// TwinCAT 3 PLC project Sample02
// ProgramVersion: 3.1.4020.10
// libraries:
//   Tc2_Standard, * (Beckhoff Automation GmbH)
//   Tc2_System, * (Beckhoff Automation GmbH)
//   Tc3_Module, * (Beckhoff Automation GmbH)
// project tree:
//   / PlcTask.TcTTO (not stored)
//   POUs/ Class Diagram.TcCD (not stored), FB_AnalogValue.TcPOU, FB_Controller.TcPOU, FB_Lamp.TcPOU, FB_LampUpDown.TcPOU, FB_LampSetDirect.TcPOU, FB_LampOnOff.TcPOU, I_Lamp.TcIO, I_Observer.TcIO, I_Subject.TcIO, MAIN.TcPOU
// real-time tasks:
//   TASK PlcTask: cycle T#10ms, priority 20, ADS port 350

// ---- POUs/I_Lamp.TcIO
INTERFACE I_Lamp

// Reduces the control value by 5 in the range of 10 to 100.
METHOD DimDown
VAR_INPUT
END_VAR
END_METHOD

// Increments the control value by 5 in the range of 10 to 100.
METHOD DimUp
VAR_INPUT
END_VAR
END_METHOD

// Sets the control value to 0.
METHOD Off
VAR_INPUT
END_VAR
END_METHOD

// Sets the control value to 100.
METHOD On
VAR_INPUT
END_VAR
END_METHOD

END_INTERFACE

// ---- POUs/I_Observer.TcIO
INTERFACE I_Observer EXTENDS __System.IQueryInterface

METHOD Update : BYTE
VAR_INPUT
	nNewValue		: BYTE(0..100);
END_VAR
END_METHOD

END_INTERFACE

// ---- POUs/I_Subject.TcIO
INTERFACE I_Subject EXTENDS __SYSTEM.IQueryInterface

METHOD Attach
VAR_INPUT
	ipObserver		: I_Observer;
END_VAR
END_METHOD

METHOD Detach
END_METHOD

END_INTERFACE

// ---- POUs/FB_AnalogValue.TcPOU
FUNCTION_BLOCK PUBLIC FB_AnalogValue IMPLEMENTS I_Observer
VAR_INPUT
END_VAR
VAR_OUTPUT
END_VAR
VAR
	_nActualValue		: BYTE(0..100);
END_VAR

PROPERTY nValue : BYTE (0..100)
GET
nValue := _nActualValue;
END_GET
END_PROPERTY

METHOD Update : BYTE
VAR_INPUT
	nNewValue		: BYTE(0..100);
END_VAR
_nActualValue := nNewValue;
END_METHOD

END_FUNCTION_BLOCK

// ---- POUs/FB_Controller.TcPOU
FUNCTION_BLOCK PUBLIC FB_Controller
VAR_INPUT
END_VAR
VAR_OUTPUT
END_VAR
VAR
	fbActualValue		: FB_AnalogValue;
	_refActiveLamp		: REFERENCE TO FB_Lamp;
END_VAR

// Reduces the control value by 5 in the range of 10 to 100.
METHOD PUBLIC DimDown
IF (__ISVALIDREF(_refActiveLamp)) THEN
	_refActiveLamp.DimDown();
END_IF
END_METHOD

// Increments the control value by 5 in the range of 10 to 100.
METHOD PUBLIC DimUp
IF (__ISVALIDREF(_refActiveLamp)) THEN
	_refActiveLamp.DimUp();
END_IF
END_METHOD

// Sets the control value to 0.
METHOD PUBLIC Off
IF (__ISVALIDREF(_refActiveLamp)) THEN
	_refActiveLamp.Off();
END_IF
END_METHOD

// Sets the control value to 100.
METHOD PUBLIC On
IF (__ISVALIDREF(_refActiveLamp)) THEN
	_refActiveLamp.On();
END_IF
END_METHOD

PROPERTY PUBLIC refActiveLamp : REFERENCE TO FB_Lamp
GET
refActiveLamp := _refActiveLamp;
END_GET
SET
IF (__ISVALIDREF(_refActiveLamp)) THEN
	_refActiveLamp.Detach();
END_IF

_refActiveLamp REF= refActiveLamp;

IF (__ISVALIDREF(refActiveLamp)) THEN
	refActiveLamp.Attach(fbActualValue);
END_IF
END_SET
END_PROPERTY

END_FUNCTION_BLOCK

// ---- POUs/FB_Lamp.TcPOU
FUNCTION_BLOCK PUBLIC ABSTRACT FB_Lamp IMPLEMENTS I_Subject, I_Lamp
VAR
	_ipObserver			: I_Observer;
END_VAR

METHOD Attach
VAR_INPUT
	ipObserver		: I_Observer;
END_VAR
IF (ipObserver = 0) THEN
	RETURN;
END_IF
_ipObserver := ipObserver;
END_METHOD

METHOD Detach
_ipObserver := 0;
END_METHOD

// Reduces the control value by 5 in the range of 10 to 100.
METHOD PUBLIC ABSTRACT DimDown
END_METHOD

// Increments the control value by 5 in the range of 10 to 100.
METHOD PUBLIC ABSTRACT DimUp
END_METHOD

// Sets the control value to 0.
METHOD PUBLIC ABSTRACT Off
END_METHOD

// Sets the control value to 100.
METHOD PUBLIC ABSTRACT On
END_METHOD

END_FUNCTION_BLOCK

// ---- POUs/FB_LampUpDown.TcPOU
FUNCTION_BLOCK PUBLIC FB_LampUpDown EXTENDS FB_Lamp
VAR
	nLightLevel			: BYTE(0..100);
END_VAR

// Reduces the control value by 5 in the range of 10 to 100.
METHOD PUBLIC DimDown
IF (nLightLevel >= 15) THEN
	OneStepDown();
	OneStepDown();
	OneStepDown();
	OneStepDown();
	OneStepDown();
END_IF
END_METHOD

// Increments the control value by 5 in the range of 10 to 100.
METHOD PUBLIC DimUp
IF (nLightLevel <= 95) THEN	
	OneStepUp();
	OneStepUp();
	OneStepUp();
	OneStepUp();
	OneStepUp();
END_IF
END_METHOD

// Sets the control value to 0.
METHOD PUBLIC Off
IF (nLightLevel > 0) THEN
	OnOff();
END_IF
END_METHOD

// Sets the control value to 100.
METHOD PUBLIC On
IF (nLightLevel = 0) THEN
	OnOff();
END_IF
END_METHOD

// Reduces the control value by 1 in the range of 10 to 100.
METHOD PUBLIC OneStepDown
nLightLevel := nLightLevel - 1;
IF (nLightLevel < 10) THEN
	nLightLevel := 10;
END_IF
IF (_ipObserver <> 0) THEN
	_ipObserver.Update(nLightLevel);
END_IF
END_METHOD

// Increments the control value by 1 in the range of 10 to 100.
METHOD PUBLIC OneStepUp
nLightLevel := nLightLevel + 1;
IF (nLightLevel > 100) THEN
	nLightLevel := 100;
END_IF
IF (_ipObserver <> 0) THEN
	_ipObserver.Update(nLightLevel);
END_IF
END_METHOD

// Toggles the control value between 0 and 100.
METHOD PUBLIC OnOff
IF (nLightLevel > 0) THEN
	nLightLevel := 0;
ELSE
	nLightLevel := 100;
END_IF
IF (_ipObserver <> 0) THEN
	_ipObserver.Update(nLightLevel);
end_IF
END_METHOD

END_FUNCTION_BLOCK

// ---- POUs/FB_LampSetDirect.TcPOU
FUNCTION_BLOCK PUBLIC FB_LampSetDirect EXTENDS FB_Lamp
VAR
	nLightLevel			: BYTE(0..100);
END_VAR

// Reduces the control value by 5 in the range of 10 to 100.
METHOD PUBLIC DimDown
IF (nLightLevel >= 15) THEN
	SetLightLevel(nLightLevel - 5);
END_IF
END_METHOD

// Increments the control value by 5 in the range of 10 to 100.
METHOD PUBLIC DimUp
IF (nLightLevel <= 95) THEN
	SetLightLevel(nLightLevel + 5);
END_IF
END_METHOD

// Sets the control value to 0.
METHOD PUBLIC Off
SetLightLevel(0);
END_METHOD

// Sets the control value to 100.
METHOD PUBLIC On
SetLightLevel(100);
END_METHOD

// Sets the control value to a value between 0 and 100.
METHOD PUBLIC SetLightLevel
VAR_INPUT
	nNewLightLevel		: BYTE(0..100);
END_VAR
nLightLevel := nNewLightLevel;
IF (_ipObserver <> 0) THEN
	_ipObserver.Update(nLightLevel);
END_IF
END_METHOD

END_FUNCTION_BLOCK

// ---- POUs/FB_LampOnOff.TcPOU
FUNCTION_BLOCK PUBLIC FB_LampOnOff EXTENDS FB_Lamp 
VAR
	nLightLevel			: BYTE(0..100);
END_VAR

// Reduces the control value by 5 in the range of 10 to 100.
METHOD PUBLIC DimDown
Off();
END_METHOD

// Increments the control value by 5 in the range of 10 to 100.
METHOD PUBLIC DimUp
On();
END_METHOD

// Sets the control value to 0.
METHOD PUBLIC Off
nLightLevel := 0;
IF (_ipObserver <> 0) THEN
	_ipObserver.Update(nLightLevel);
END_IF
END_METHOD

// Sets the control value to 100.
METHOD PUBLIC On
nLightLevel := 100;
IF (_ipObserver <> 0) THEN
	_ipObserver.Update(nLightLevel);
END_IF
END_METHOD

END_FUNCTION_BLOCK

// ---- POUs/MAIN.TcPOU
PROGRAM MAIN
VAR
	fbController		: FB_Controller();
	fbLampOnOff			: FB_LampOnOff();
	fbLampSetDirect		: FB_LampSetDirect();
	fbLampUpDown		: FB_LampUpDown();
	nSetLamp			: INT;
	bDimUp, bDimDown	: BOOL;
	bOff, bOn			: BOOL;
END_VAR

CASE nSetLamp OF
	1:
		fbController.refActiveLamp REF= fbLampOnOff;
		nSetLamp := 0;
	2:
		fbController.refActiveLamp REF= fbLampSetDirect;
		nSetLamp := 0;
	3:
		fbController.refActiveLamp REF= fbLampUpDown;
		nSetLamp := 0;
END_CASE

IF (bDimUp) THEN
	fbController.DimUp();
	bDimUp := FALSE;
END_IF

IF (bDimDown) THEN
	fbController.DimDown();
	bDimDown := FALSE;
END_IF

IF (bOff) THEN
	fbController.Off();
	bOff := FALSE;
END_IF

IF (bOn) THEN
	fbController.On();
	bOn := FALSE;
END_IF

END_PROGRAM
